{attribute addProperty BoxType "EL3773-0000-0018"}
{attribute addProperty Id "I3_StatusAT %I*I3_Status_E2EFACF1162"}
{attribute addProperty CRC "2391859512"}
{attribute addProperty SizeInBites "16"}
{attribute addProperty SizeInBytes "2"}
TYPE L3_Current_Status_8E90E138 :
STRUCT
	{attribute addProperty Name "I3_Status"}
	I3_Status AT %I* : I3_Status_E2EFACF1;
END_STRUCT
END_TYPE

(* stored: Version 1.2.0.0, ProductVersion 3.1.4024.9
   DUT L3_Current_Status_8E90E138: Id {3c888885-a4ad-4ebd-b9ea-4ef0beae981c} *)
